// TIA Portal V17 export
// export: Created 2022-02-03T14:45:12.9399388Z, ExportSetting WithDefaults, DisplayName Totally Integrated Automation Portal, DisplayVersion V17, DisplayName TIA Portal Openness, DisplayVersion V17, DisplayName TIA Portal Version Control Interface, DisplayVersion V17, DisplayName SINAMICS Startdrive Advanced, DisplayVersion V17, DisplayName SINAMICS Startdrive G130, G150, S120, S150, SINAMICS MV, S210, DisplayVersion V17, DisplayName SINAMICS Startdrive G110M, G120, G120C, G120D, G120P, G115D, DisplayVersion V17, DisplayName STEP 7 Professional, DisplayVersion V17, DisplayName STEP 7 Safety, DisplayVersion V17, DisplayName WinCC Advanced, DisplayVersion V17
FUNCTION_BLOCK "NewWeightToStore"   // FB7, LAD
VERSION : 0.1
// stored: Access Published, AutoNumber true, IsIECCheckEnabled false, IsRetainMemResEnabled false, MemoryReserve 100, SetENOAutomatically false, UDAEnableTagReadback false
   VAR_INPUT
      occupiedBay : Array["FIRSTBAY".."LASTBAY"] of Bool;
      weightBay : Array["FIRSTBAY".."LASTBAY"] of UInt;
      initStore : Bool;
      storeNo : UInt;
      initAllStores : Bool;
   END_VAR
   VAR_OUTPUT
      storeFull : Bool;
   END_VAR
   VAR_IN_OUT
      store : Array[0..9] of "typeStore";
      storeStatistics : "typeStoreStatistics";
   END_VAR
   VAR
      statOldOccupiedBay : Array["FIRSTBAY".."LASTBAY"] of Bool;
      statOldInitStore : Bool;
      statStoreNo : UInt;
   END_VAR
   VAR_TEMP   // added for the SCL form of the ladder/FBD networks
      _w1 : Bool;
      _w2 : Bool;
      _w3 : Bool;
   END_VAR
BEGIN

REGION Network 1
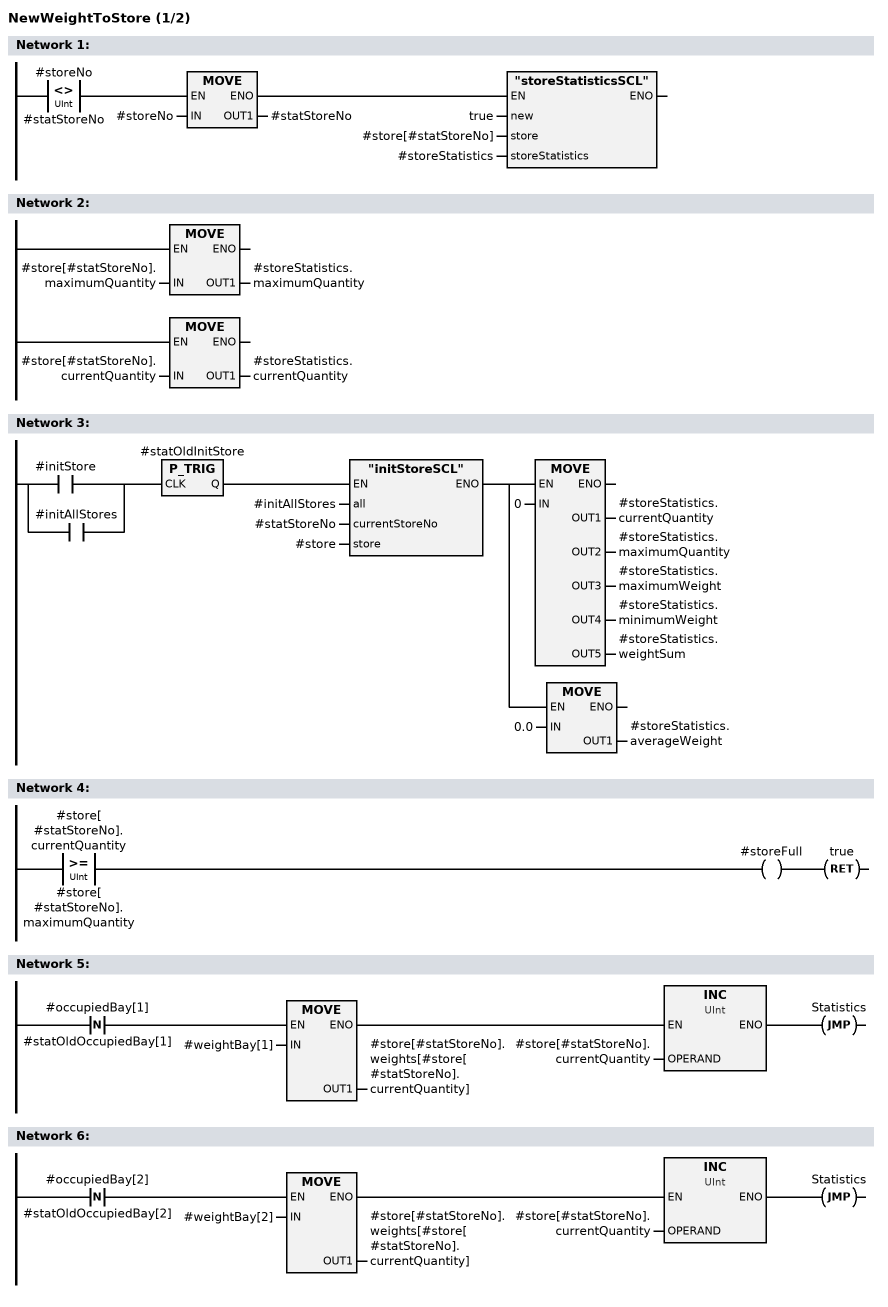
   RUNG wire#powerrail
      { S7_Templates := "SrcType := UInt" } NE_Contact(in1 := #storeNo, in2 := #statStoreNo)
      Move(in := #storeNo, out1 => #statStoreNo)
      "storeStatisticsSCL"(new := true, store := #store[#statStoreNo], storeStatistics := #storeStatistics)
   END_RUNG
   // the same network as SCL:
   #_w1 := #storeNo <> #statStoreNo;
   IF #_w1 THEN
       #statStoreNo := #storeNo;
       "storeStatisticsSCL"(new := true, store := #store[#statStoreNo], storeStatistics := #storeStatistics);
   END_IF;
END_REGION

REGION Network 2
   RUNG wire#powerrail
      Move(in := #store[#statStoreNo].maximumQuantity, out1 => #storeStatistics.maximumQuantity)
   END_RUNG
   RUNG wire#powerrail
      Move(in := #store[#statStoreNo].currentQuantity, out1 => #storeStatistics.currentQuantity)
   END_RUNG
   // the same network as SCL:
   #storeStatistics.maximumQuantity := #store[#statStoreNo].maximumQuantity;
   #storeStatistics.currentQuantity := #store[#statStoreNo].currentQuantity;
END_REGION

REGION Network 3
   RUNG wire#powerrail
      Contact( #initStore )
      wire#w1
      P_Trig( #statOldInitStore )
      "initStoreSCL"(all := #initAllStores, currentStoreNo := #statStoreNo, store := #store)
      wire#w2
      Move(in := 0, out1 => #storeStatistics.currentQuantity, out2 => #storeStatistics.maximumQuantity, out3 => #storeStatistics.maximumWeight, out4 => #storeStatistics.minimumWeight, out5 => #storeStatistics.weightSum)
   END_RUNG
   RUNG wire#powerrail
      Contact( #initAllStores )
   END_RUNG wire#w1
   RUNG wire#w2
      Move(in := 0.0, out1 => #storeStatistics.averageWeight)
   END_RUNG
   // the same network as SCL:
   #_w1 := #initStore OR #initAllStores;
   #_w2 := #_w1 AND NOT #statOldInitStore;   // rising edge
   #statOldInitStore := #_w1;
   "initStoreSCL"(EN := #_w2,
                  all := #initAllStores,
                  currentStoreNo := #statStoreNo,
                  store := #store,
                  ENO => #_w3);
   IF #_w3 THEN
       #storeStatistics.currentQuantity := 0;
       #storeStatistics.maximumQuantity := 0;
       #storeStatistics.maximumWeight := 0;
       #storeStatistics.minimumWeight := 0;
       #storeStatistics.weightSum := 0;
       #storeStatistics.averageWeight := 0.0;
   END_IF;
END_REGION

REGION Network 4
   #storeFull := #store[#statStoreNo].currentQuantity >= #store[#statStoreNo].maximumQuantity;
   IF #storeFull THEN
       ENO := true;
       RETURN;
   END_IF;
END_REGION

REGION Network 5
   RUNG wire#powerrail
      N_Contact(operand := #occupiedBay[1], bit := #statOldOccupiedBay[1])
      Move(in := #weightBay[1], out1 => #store[#statStoreNo].weights[#store[#statStoreNo].currentQuantity])
      { S7_Templates := "DestType := UInt" } Inc( #store[#statStoreNo].currentQuantity )
      JumpCoil( Statistics )
   END_RUNG
   // the same network as SCL:
   #_w1 := NOT #occupiedBay[1] AND #statOldOccupiedBay[1];   // falling edge of #occupiedBay[1]
   #statOldOccupiedBay[1] := #occupiedBay[1];
   IF #_w1 THEN
       #store[#statStoreNo].weights[#store[#statStoreNo].currentQuantity] := #weightBay[1];
       #store[#statStoreNo].currentQuantity := #store[#statStoreNo].currentQuantity + 1;
       GOTO Statistics;
   END_IF;
END_REGION

REGION Network 6
   RUNG wire#powerrail
      N_Contact(operand := #occupiedBay[2], bit := #statOldOccupiedBay[2])
      Move(in := #weightBay[2], out1 => #store[#statStoreNo].weights[#store[#statStoreNo].currentQuantity])
      { S7_Templates := "DestType := UInt" } Inc( #store[#statStoreNo].currentQuantity )
      JumpCoil( Statistics )
   END_RUNG
   // the same network as SCL:
   #_w1 := NOT #occupiedBay[2] AND #statOldOccupiedBay[2];   // falling edge of #occupiedBay[2]
   #statOldOccupiedBay[2] := #occupiedBay[2];
   IF #_w1 THEN
       #store[#statStoreNo].weights[#store[#statStoreNo].currentQuantity] := #weightBay[2];
       #store[#statStoreNo].currentQuantity := #store[#statStoreNo].currentQuantity + 1;
       GOTO Statistics;
   END_IF;
END_REGION

REGION Network 7
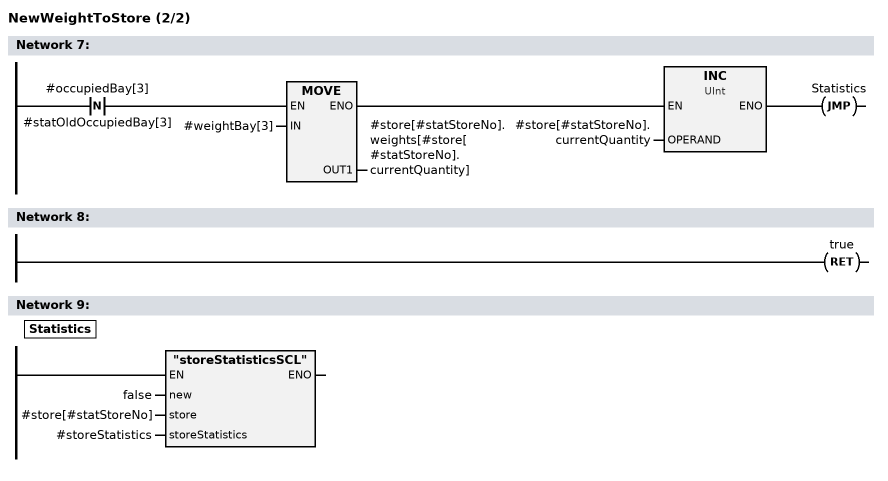
   RUNG wire#powerrail
      N_Contact(operand := #occupiedBay[3], bit := #statOldOccupiedBay[3])
      Move(in := #weightBay[3], out1 => #store[#statStoreNo].weights[#store[#statStoreNo].currentQuantity])
      { S7_Templates := "DestType := UInt" } Inc( #store[#statStoreNo].currentQuantity )
      JumpCoil( Statistics )
   END_RUNG
   // the same network as SCL:
   #_w1 := NOT #occupiedBay[3] AND #statOldOccupiedBay[3];   // falling edge of #occupiedBay[3]
   #statOldOccupiedBay[3] := #occupiedBay[3];
   IF #_w1 THEN
       #store[#statStoreNo].weights[#store[#statStoreNo].currentQuantity] := #weightBay[3];
       #store[#statStoreNo].currentQuantity := #store[#statStoreNo].currentQuantity + 1;
       GOTO Statistics;
   END_IF;
END_REGION

REGION Network 8
   ENO := true;
   RETURN;
END_REGION

REGION Network 9
   Label( Statistics )
   RUNG wire#powerrail
      "storeStatisticsSCL"(new := false, store := #store[#statStoreNo], storeStatistics := #storeStatistics)
   END_RUNG
   // the same network as SCL:
   Statistics:
   "storeStatisticsSCL"(new := false, store := #store[#statStoreNo], storeStatistics := #storeStatistics);
END_REGION
END_FUNCTION_BLOCK
